FUNCTION_BLOCK FB_Sensor EXTENDS FB_SensorBase
VAR_INPUT
END_VAR
VAR_OUTPUT
END_VAR
VAR
	bSensor_HardwareInput	AT %I* : BOOL;	//Hardware input bit from the hysical sensor
END_VAR

METHOD PRIVATE HardwareUpdate : BOOL
VAR_INPUT
END_VAR
SUPER^.HardwareUpdate();

bRawSensorInput := bSensor_HardwareInput;
END_METHOD

END_FUNCTION_BLOCK

(* stored: Version 1.1.0.1, ProductVersion 3.1.4024.9
   POU FB_Sensor: Id {600a0be8-8f86-40d7-91ca-048d45e1e72d}, SpecialFunc None
   Folder 01_SUPER_Overrides: Id {0678f6d0-782c-4a6f-9d10-9b0a34b9542e}
   Method HardwareUpdate: Id {10f795a8-9ec4-4b2a-8124-c7a53d3ba7ea} *)
